# EPICS alarm handler configuration: epics_alh/alarms_list_TargetDAQ.alhConfig
GROUP NULL TargetDAQ

GROUP TargetDAQ CRYO

GROUP CRYO Insert
CHANNEL Insert INS_T01
CHANNEL Insert INS_T02
CHANNEL Insert INS_T03
CHANNEL Insert INS_T04
CHANNEL Insert INS_T05

GROUP CRYO Fridge

GROUP Fridge T
CHANNEL T EVF_T01
CHANNEL T EVF_T02
CHANNEL T EVF_T03
CHANNEL T EVF_T04
CHANNEL T EVF_T05
CHANNEL T EVF_T06
CHANNEL T EVF_T07
CHANNEL T EVF_T08

GROUP Fridge P
CHANNEL P EVF_P01
CHANNEL P EVF_P02
CHANNEL P EVF_P03

GROUP Fridge F
CHANNEL F EVF_F01
CHANNEL F EVF_FS1
CHANNEL F EVF_F02

GROUP Fridge L
CHANNEL L EVF_L01
CHANNEL L EVF_LS1

GROUP Fridge S
CHANNEL S EVF_S01
CHANNEL S EVF_SS1
CHANNEL S EVF_S02
CHANNEL S EVF_S03
CHANNEL S EVF_SS3
CHANNEL S EVF_S04

GROUP CRYO Roots

GROUP Roots T
CHANNEL T RPS_T01
CHANNEL T RPS_T02
CHANNEL T RPS_T03

GROUP Roots P
CHANNEL P RPS_P01
CHANNEL P RPS_P02
CHANNEL P RPS_P03
CHANNEL P RPS_P04
CHANNEL P RPS_P05
CHANNEL P RPS_P06

GROUP Roots F
CHANNEL F RPS_F01
CHANNEL F RPS_F02
CHANNEL F RPS_F03
CHANNEL F RPS_F04
CHANNEL F RPS_F05
CHANNEL F RPS_F06

GROUP CRYO Vacuum
CHANNEL Vacuum OVS_P01
CHANNEL Vacuum OVS_P02

GROUP CRYO WarmGas

GROUP TargetDAQ MAGNET

GROUP MAGNET T
CHANNEL T SCM_T01
CHANNEL T SCM_T02
CHANNEL T SCM_T03
CHANNEL T SCM_T04
CHANNEL T SCM_T05
CHANNEL T SCM_T06
CHANNEL T SCM_T07
CHANNEL T SCM_T08
CHANNEL T SCM_T09
CHANNEL T SCM_T10
CHANNEL T SCM_T11
CHANNEL T SCM_T12

GROUP MAGNET F
CHANNEL F SCM_F01
CHANNEL F SCM_F02

GROUP MAGNET L
CHANNEL L SCM_L01
CHANNEL L SCM_L02

GROUP MAGNET IVB
CHANNEL IVB SCM_I01
CHANNEL IVB SCM_IS1
CHANNEL IVB SCM_R01
CHANNEL IVB SCM_RS1
CHANNEL IVB SCM_V01
CHANNEL IVB SCM_B01

GROUP MAGNET STATE
CHANNEL STATE SCM_MOD
CHANNEL STATE SCM_MST
CHANNEL STATE SCM_HST
CHANNEL STATE SCM_SST
CHANNEL STATE SCM_SMD

GROUP TargetDAQ u-WAVE

GROUP u-WAVE T
CHANNEL T MWS_T01
CHANNEL T MWS_T02
CHANNEL T MWS_T03
CHANNEL T MWS_T04

GROUP u-WAVE S
CHANNEL S MWS_S01
CHANNEL S MWS_SS1
CHANNEL S MWS_S02
CHANNEL S MWS_S03

GROUP u-WAVE PARM
CHANNEL PARM MWS_uWF
CHANNEL PARM MWS_uWP
CHANNEL PARM MWS_V01
CHANNEL PARM MWS_V02
CHANNEL PARM MWS_V03
CHANNEL PARM MWS_I01
CHANNEL PARM MWS_I02
CHANNEL PARM MWS_STA
CHANNEL PARM MWS_FMF
CHANNEL PARM MWS_FMA
CHANNEL PARM MWS_FMO

GROUP TargetDAQ LIFTER
CHANNEL LIFTER TMS_S01
CHANNEL LIFTER TMS_SS1
CHANNEL LIFTER TMS_S02
CHANNEL LIFTER TMS_S03
CHANNEL LIFTER TMS_S04
CHANNEL LIFTER TMS_S05
CHANNEL LIFTER TMS_S06
CHANNEL LIFTER TMS_S07
CHANNEL LIFTER TMS_S08

GROUP TargetDAQ NMR
